// TIA Portal V16 export
// export: Created 2021-11-12T13:31:55.260915Z, ExportSetting WithDefaults, DisplayName Totally Integrated Automation Portal, DisplayVersion V16 Update 3, DisplayName TIA Portal Version Control Interface, DisplayVersion V16 Update 2, DisplayName TIA Portal Openness, DisplayVersion V16 Update 3, DisplayName SINAMICS Startdrive Advanced, DisplayVersion V16 Update 5, DisplayName SINAMICS Startdrive G130, G150, S120, S150, SINAMICS MV, S210, DisplayVersion V16 Update 5, DisplayName SINAMICS Startdrive G110M, G120, G120C, G120D, G120P, G115D, DisplayVersion V16 Update 5, DisplayName STEP 7 Professional, DisplayVersion V16 Update 3, DisplayName STEP 7 Safety, DisplayVersion V16, DisplayName WinCC UA Professional, DisplayVersion V16 Update 3
DATA_BLOCK "HMI_CMD_000+UC10"   // DB159
{ S7_Optimized_Access := 'TRUE' }
VERSION : 0.1
// stored: AutoNumber true, DBAccessibleFromOPCUA true, IsOnlyStoredInLoadMemory false, IsRetainMemResEnabled false, IsWriteProtectedInAS false, MemoryReserve 100
   VAR
      xxxxx___BinarySensors___xxxxx : Byte;
      xxxxx___BinaryOthers___xxxxx : Byte;
      FV01_11 { S7_SetPoint := 'True'} : "UDT_CH_DI_Command";   // Přepěťová ochrana OK
      FB21_14 { S7_SetPoint := 'True'} : "UDT_CH_DI_Command";   // 230V Osvětlení rozvaděče se zásuvkou je OK
      FC21_14 { S7_SetPoint := 'True'} : "UDT_CH_DI_Command";   // 230V Chlazeni rozvaděče je OK
      EC01_3 { S7_SetPoint := 'True'} : "UDT_CH_DI_Command";   // Chlazení rozvaděče je OK
      FC01_14 { S7_SetPoint := 'True'} : "UDT_CH_DI_Command";   // 400V Napájení 24V DC je OK
      TB01_14 { S7_SetPoint := 'True'} : "UDT_CH_DI_Command";   // Napájení 24V DC je OK
      FC30_14 { S7_SetPoint := 'True'} : "UDT_CH_DI_Command";   // 24V Distribuce je OK
      FC30_24 { S7_SetPoint := 'True'} : "UDT_CH_DI_Command";   // 24V Distribuce 90 >% zatížení
      FC50_14 { S7_SetPoint := 'True'} : "UDT_CH_DI_Command";   // 24V Distribuce je OK
      FC51_24 { S7_SetPoint := 'True'} : "UDT_CH_DI_Command";   // 24V Distribuce 90 >% zatížení
      "UC12-FC21_14" { S7_SetPoint := 'True'} : "UDT_CH_DI_Command";   // 230V Chlazeni rozvaděče je OK
      "UC12-EC01_3" { S7_SetPoint := 'True'} : "UDT_CH_DI_Command";   // Chlazení rozvaděče je OK
      "UC11-FC01_14" { S7_SetPoint := 'True'} : "UDT_CH_DI_Command";   // 400V Čerpadlo ponorné P51 OK
      "UC11-FC02_14" { S7_SetPoint := 'True'} : "UDT_CH_DI_Command";   // 400V Čerpadlo ponorné P52 OK
      "UC11-FC03_14" { S7_SetPoint := 'True'} : "UDT_CH_DI_Command";   // 400V Čerpadlo ponorné P61 OK
      xxxxx___AnalogueSensors___xxxxx : Byte;
      xxxxx___Drives___xxxxx : Byte;
      xxxxx___Other___xxxxx : Byte;
      xxxxx___Alarms___xxxxx : Byte;
      FV01_12 { S7_SetPoint := 'True'} : "UDT_DI_Mon_Command";   // Přepěťová ochrana OK
      FB21_15 { S7_SetPoint := 'True'} : "UDT_DI_Mon_Command";   // 230V Osvětlení rozvaděče se zásuvkou je OK
      FC21_15 { S7_SetPoint := 'True'} : "UDT_DI_Mon_Command";   // 230V Chlazeni rozvaděče je OK
      EC01_4 { S7_SetPoint := 'True'} : "UDT_DI_Mon_Command";   // Chlazení rozvaděče je OK
      FC01_15 { S7_SetPoint := 'True'} : "UDT_DI_Mon_Command";   // 400V Napájení 24V DC je OK
      TB01_15 { S7_SetPoint := 'True'} : "UDT_DI_Mon_Command";   // Napájení 24V DC je OK
      FC30_15 { S7_SetPoint := 'True'} : "UDT_DI_Mon_Command";   // 24V Distribuce je OK
      FC30_25 { S7_SetPoint := 'True'} : "UDT_DI_Mon_Command";   // 24V Distribuce 90 >% zatížení
      FC50_15 { S7_SetPoint := 'True'} : "UDT_DI_Mon_Command";   // 24V Distribuce je OK
      FC51_25 { S7_SetPoint := 'True'} : "UDT_DI_Mon_Command";   // 24V Distribuce 90 >% zatížení
      "UC12-FC21_15" { S7_SetPoint := 'True'} : "UDT_DI_Mon_Command";   // 230V Chlazeni rozvaděče je OK
      "UC12-EC01_4" { S7_SetPoint := 'True'} : "UDT_DI_Mon_Command";   // Chlazení rozvaděče je OK
      "UC11-FC01_15" { S7_SetPoint := 'True'} : "UDT_DI_Mon_Command";   // 400V Čerpadlo ponorné P51 OK
      "UC11-FC02_15" { S7_SetPoint := 'True'} : "UDT_DI_Mon_Command";   // 400V Čerpadlo ponorné P52 OK
      "UC11-FC03_15" { S7_SetPoint := 'True'} : "UDT_DI_Mon_Command";   // 400V Čerpadlo ponorné P61 OK
   END_VAR
BEGIN
END_DATA_BLOCK
